// TIA Portal V17 export
// export: Created 2022-03-12T16:05:30.2217505Z, ExportSetting WithDefaults, DisplayName Totally Integrated Automation Portal, DisplayVersion V17, DisplayName TIA Portal Openness, DisplayVersion V17, DisplayName TIA Portal Version Control Interface, DisplayVersion V17, DisplayName STEP 7 Professional, DisplayVersion V17, DisplayName STEP 7 Safety, DisplayVersion V17, DisplayName WinCC Advanced / Unified PC, DisplayVersion V17
DATA_BLOCK "HMI_Data"   // DB31615
TITLE = CPG_HMI_Data
{ S7_Optimized_Access := 'TRUE' }
AUTHOR : tech.team.motioncontrol@siemens.com
FAMILY : CPG
VERSION : 1.0
// Support: tech.team.motioncontrol@siemens.com
// Fax: +49 (0) 9131/98-1297
// stored: AutoNumber true, DBAccessibleFromOPCUA true, DBAccessibleFromWebserver true, IsOnlyStoredInLoadMemory false, IsRetainMemResEnabled false, IsWriteProtectedInAS false, MemoryReserve 0
   VAR
      resetPackMLTimers : Bool;   // Reset the PackML Timer values when set (1).
   END_VAR
   VAR RETAIN
      languageSelected : Int;   // This is the value of the language selected in the HMI (0=English, 1=DE, 2=SP, 3
   END_VAR
   VAR
      modeCurrentTime { ExternalWritable := 'False'} : DInt;   // Time spent in the current mode [seconds](reset each time new mode is entered)
      modeCumulativeTime { ExternalWritable := 'False'} : DInt;   // Accumulative Time spent in the current mode [seconds]
      State_Current_Times { ExternalWritable := 'False'} : Array[0.."LPMLV30_STATES_UPPER_LIM"] of DInt;   // Current Time (# of seconds) spent for each state for active mode.
      State_Cumulative_Times { ExternalWritable := 'False'} : Array[0.."LPMLV30_STATES_UPPER_LIM"] of DInt;   // Accumulative Time (# of seconds) spent for each state for active mode.
      alarmSortedList { ExternalWritable := 'False'; S7_SetPoint := 'True'} : Array[0.."CPG_NO_OF_HMI_SORT_EVENTS_UPPER_LIM"] of "CPG_typeEvent";   // Alarm Sorted List for HMI - summary of Active Events
      EM_SortDisable_Alarm : Struct   // Alarm Disable for Equipment Modules (EMs)
         Unit : Bool;   // If bool is reset, then Unit sort filter is enabled, else it's disabled.
         EM00 : Bool;   // If bool is reset, then EMxx sort filter is enabled, else it's disabled.
         EM01 : Bool;   // If bool is reset, then EMxx sort filter is enabled, else it's disabled.
         EM02 : Bool;   // If bool is reset, then EMxx sort filter is enabled, else it's disabled.
         EM03 : Bool;   // If bool is reset, then EMxx sort filter is enabled, else it's disabled.
         EM04 : Bool;   // If bool is reset, then EMxx sort filter is enabled, else it's disabled.
         EM05 : Bool;   // If bool is reset, then EMxx sort filter is enabled, else it's disabled.
         EM06 : Bool;   // If bool is reset, then EMxx sort filter is enabled, else it's disabled.
         EM07 : Bool;   // If bool is reset, then EMxx sort filter is enabled, else it's disabled.
         EM08 : Bool;   // If bool is reset, then EMxx sort filter is enabled, else it's disabled.
         EM09 : Bool;   // If bool is reset, then EMxx sort filter is enabled, else it's disabled.
         EM10 : Bool;   // If bool is reset, then EMxx sort filter is enabled, else it's disabled.
      END_STRUCT;
      alarmFilter { S7_SetPoint := 'True'} : "CPG_typeSortFilter";   // HMI Commands to control the Alarm Sort Filter
      warningSortedList { ExternalWritable := 'False'; S7_SetPoint := 'True'} : Array[0.."CPG_NO_OF_HMI_SORT_EVENTS_UPPER_LIM"] of "CPG_typeEvent";   // Warning Sorted List for HMI - summary of Active Events
      EMSortDisableWarning : Struct   // Warning Disable for Equipment Modules (EMs)
         Unit : Bool;   // If bool is reset, then Unit sort filter is enabled, else it's disabled.
         EM00 : Bool;   // If bool is reset, then EMxx sort filter is enabled, else it's disabled.
         EM01 : Bool;   // If bool is reset, then EMxx sort filter is enabled, else it's disabled.
         EM02 : Bool;   // If bool is reset, then EMxx sort filter is enabled, else it's disabled.
         EM03 : Bool;   // If bool is reset, then EMxx sort filter is enabled, else it's disabled.
         EM04 : Bool;   // If bool is reset, then EMxx sort filter is enabled, else it's disabled.
         EM05 : Bool;   // If bool is reset, then EMxx sort filter is enabled, else it's disabled.
         EM06 : Bool;   // If bool is reset, then EMxx sort filter is enabled, else it's disabled.
         EM07 : Bool;   // If bool is reset, then EMxx sort filter is enabled, else it's disabled.
         EM08 : Bool;   // If bool is reset, then EMxx sort filter is enabled, else it's disabled.
         EM09 : Bool;   // If bool is reset, then EMxx sort filter is enabled, else it's disabled.
         EM10 : Bool;   // If bool is reset, then EMxx sort filter is enabled, else it's disabled.
      END_STRUCT;
      WarningFilter { S7_SetPoint := 'True'} : "CPG_typeSortFilter";   // HMI Commands to control the Warning Sort Filter
      HMIWarningMsgScroll { ExternalWritable := 'False'} : String[40];   // Warning Message - scroll of all active warnings
      ModeNames { ExternalWritable := 'False'} : Array[0.."LPMLV30_MODES_UPPER_LIM"] of String[18];   // Mode Names for selected language
      StateNames { ExternalWritable := 'False'} : Array[0.."LPMLV30_STATES_UPPER_LIM"] of String[16];   // State Names for selectecd modes
      PLCDateTime { ExternalWritable := 'False'} : Struct   // Date Time for WinCC Flexible HMI format
         DATE_TIME { ExternalWritable := 'False'} : Date_And_Time := DT#12-7-12-18:16:34.356;   // Current Time and Date of PLC
         reserve { ExternalWritable := 'False'} : Array[0..3] of Byte;   // Filler bytes used to sync HMI clock with PLC clock. Do not change.
      END_STRUCT;
      diagnosticsBufferIndexForHMI { ExternalWritable := 'False'} : Int;   // Diagnostics to HMI
      diagnosticsBufferEntryForHMI { ExternalWritable := 'False'; S7_SetPoint := 'True'} : "typeLPMLV30_DiagnosticsEntry";   // Diagnostics to HMI
      HMICoordination { ExternalWritable := 'False'} : Word;   // HMI Coordination area pointer: Bit0 = Startup; 1=OpMode (0=on, 1=off-line), 2=life bit
      HMICurrentScreenID : Int;   // HMI Current screen number
      CMDs : Struct   // HMI Commands
         PB_Start : Bool;   // HMI Push Button Command - Start
         PB_Stop : Bool;   // HMI Push Button Command - Stop
         PB_Hold : Bool;   // HMI Push Button Command - Hold
         PB_Reset : Bool;   // HMI Push Button Command - Reset
         PB_Complete : Bool;   // HMI Push Button Command - Complete (demo purposes only)
         PB_EStop : Bool;   // HMI Push Button Command - EStop (demo purposes only)
         PB_Abort : Bool;   // HMI Push Button Command - Abort (demo purposes only)
         PB_ProdSimulate : Bool;   // HMI Push Button Command - Product Simulate Enable (demo purposes only)
         PB_DriveSimulate : Bool;   // HMI Push Button Command - Drive / Axis Simulate (demo purposes only)
      END_STRUCT;
   END_VAR
BEGIN
END_DATA_BLOCK
